// TIA Portal V17 export
// export: Created 2025-01-08T13:55:33.962402Z, ExportSetting WithDefaults, DisplayName Totally Integrated Automation Portal, DisplayVersion V17, DisplayName TIA Portal Openness, DisplayVersion V17, DisplayName TIA Portal Version Control Interface, DisplayVersion V17, DisplayName SINAMICS Startdrive Advanced, DisplayVersion V17 Update2, DisplayName SINAMICS Startdrive G130, G150, S120, S150, SINAMICS MV, S210, DisplayVersion V17 Update2, DisplayName SINAMICS Startdrive G110M, G120, G120C, G120D, G120P, G115D, DisplayVersion V17 Update2, DisplayName STEP 7 Professional, DisplayVersion V17, DisplayName STEP 7 Safety, DisplayVersion V17, DisplayName WinCC Advanced, DisplayVersion V17
DATA_BLOCK "FB_Com_DB"   // DB3
VERSION : 0.1
// stored: AutoNumber true, DBAccessibleFromOPCUA true, DBAccessibleFromWebserver true, InstanceOfName FB_Com, InstanceOfType FB
"FB_Com"
   // VAR
   //    TRCV_C_Instance { S7_SetPoint := 'True'} : TRCV_C;
   //    GET_Instance { S7_SetPoint := 'True'} : GET;
   //    TRCV_C_Instance_1 { S7_SetPoint := 'True'} : TRCV_C;
   //    Diff : LInt;
   // END_VAR
BEGIN
END_DATA_BLOCK
